FUNCTION_BLOCK SchieberVerriegelung (* Template for a Basic Function Block Type *)
  (* Standard: 61499-2; Description: Copyright (c) 2025 HR Agrartechnik GmbH This program and the accompanying materials are made available under the terms of the Eclipse Public License 2.0 which is available at https://www.eclipse.org/legal/epl-2.0/ SPDX-License-Identifier: EPL-2.0 *)
  (* Version 1.0, 2025-06-04, Franz Höpfinger, HR Agrartechnik GmbH *)
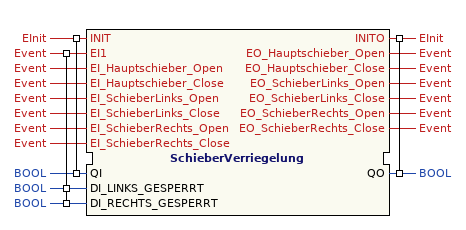
  EVENT_INPUT
    INIT : EInit WITH QI; (* Initialization Request *)
    EI1 WITH DI_LINKS_GESPERRT, DI_RECHTS_GESPERRT;
    EI_Hauptschieber_Open;
    EI_Hauptschieber_Close;
    EI_SchieberLinks_Open;
    EI_SchieberLinks_Close;
    EI_SchieberRechts_Open;
    EI_SchieberRechts_Close;
  END_EVENT
  EVENT_OUTPUT
    INITO : EInit WITH QO; (* Initialization Confirm *)
    EO_Hauptschieber_Open;
    EO_Hauptschieber_Close;
    EO_SchieberLinks_Open;
    EO_SchieberLinks_Close;
    EO_SchieberRechts_Open;
    EO_SchieberRechts_Close;
  END_EVENT
  VAR_INPUT
    QI : BOOL; (* Input event qualifier *)
    DI_LINKS_GESPERRT : BOOL;
    DI_RECHTS_GESPERRT : BOOL;
  END_VAR
  VAR_OUTPUT
    QO : BOOL; (* Output event qualifier *)
  END_VAR
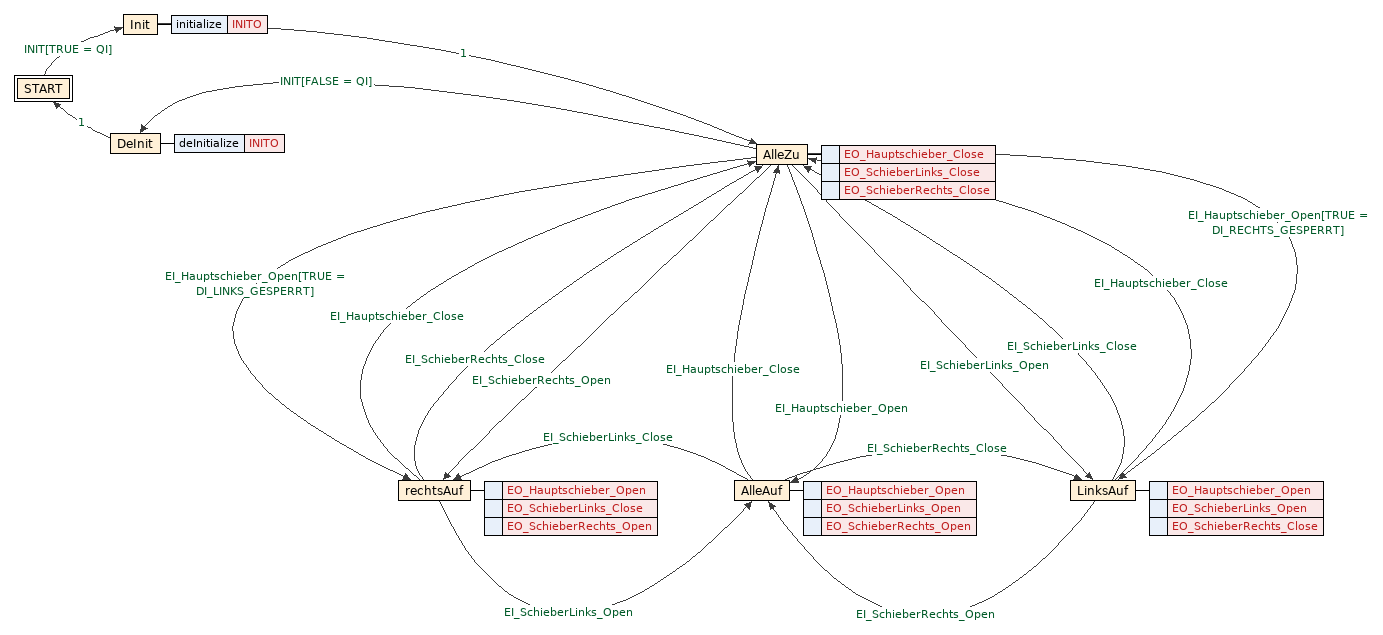
  EC_STATES
    START; (* Initial State *)
    Init : initialize -> INITO; (* Initialization *)
    DeInit : deInitialize -> INITO;
    AlleZu : -> EO_Hauptschieber_Close, -> EO_SchieberLinks_Close, -> EO_SchieberRechts_Close;
    AlleAuf : -> EO_Hauptschieber_Open, -> EO_SchieberLinks_Open, -> EO_SchieberRechts_Open;
    LinksAuf : -> EO_Hauptschieber_Open, -> EO_SchieberLinks_Open, -> EO_SchieberRechts_Close;
    rechtsAuf : -> EO_Hauptschieber_Open, -> EO_SchieberLinks_Close, -> EO_SchieberRechts_Open;
  END_STATES
  EC_TRANSITIONS
    START TO Init := INIT[TRUE = QI];
    DeInit TO START := 1;
    AlleZu TO rechtsAuf := EI_SchieberRechts_Open;
    AlleZu TO LinksAuf := EI_SchieberLinks_Open;
    rechtsAuf TO AlleZu := EI_SchieberRechts_Close;
    LinksAuf TO AlleZu := EI_SchieberLinks_Close;
    LinksAuf TO AlleAuf := EI_SchieberRechts_Open;
    rechtsAuf TO AlleAuf := EI_SchieberLinks_Open;
    AlleAuf TO rechtsAuf := EI_SchieberLinks_Close;
    AlleAuf TO LinksAuf := EI_SchieberRechts_Close;
    AlleAuf TO AlleZu := EI_Hauptschieber_Close;
    rechtsAuf TO AlleZu := EI_Hauptschieber_Close;
    LinksAuf TO AlleZu := EI_Hauptschieber_Close;
    AlleZu TO DeInit := INIT[FALSE = QI];
    Init TO AlleZu := 1;
    AlleZu TO LinksAuf := EI_Hauptschieber_Open[TRUE = DI_RECHTS_GESPERRT];
    AlleZu TO rechtsAuf := EI_Hauptschieber_Open[TRUE = DI_LINKS_GESPERRT];
    AlleZu TO AlleAuf := EI_Hauptschieber_Open;
  END_TRANSITIONS
  ALGORITHM initialize IN ST: (* Initialization algorithm *)
QO := QI;
  END_ALGORITHM
  ALGORITHM deInitialize IN ST: (* Normally executed algorithm *)
QO := FALSE;
  END_ALGORITHM
  ALGORITHM normalOperation IN ST: (* new algorithm *)
QO := QI;

IF TRUE  = QI THEN
  (*  only perform normal operation of QI is true*)

END_IF;
  END_ALGORITHM
END_FUNCTION_BLOCK
